PROGRAM EM8000
VAR	
	_control	: StewartControl;
	UdpIO		: UdpClient(3232258590, 50030, 50040, SIZEOF(_control), ADR(_control), SIZEOF(feedback), ADR(feedback));
	
	Pi 			: REAL := 3.141592653589793;
END_VAR

VAR_INPUT
	control		: StewartControl;
END_VAR

VAR_OUTPUT
	feedback	: StewartFeedback;
END_VAR



// Assign c0ntrol to local _control
_control.CMND := control.CMND;

// Addd maximum limit to udp input _control
_control.X_EXTRA 		:= LIMIT(-0.6, control.X_EXTRA, 0.6);
_control.Y_EXTRA 		:= LIMIT(-0.6, control.Y_EXTRA, 0.6);
_control.Z_EXTRA 		:= LIMIT(-0.6, control.Z_EXTRA, 0.6);

_control.PSI_EXTRA 		:= LIMIT(-10.0/180.0*Pi, control.PSI_EXTRA, 10.0/180.0*Pi);
_control.THETA_EXTRA 	:= LIMIT(-10.0/180.0*Pi, control.THETA_EXTRA, 10.0/180.0*Pi);
_control.PHI_EXTRA 		:= LIMIT(-10.0/180.0*Pi, control.PHI_EXTRA, 10.0/180.0*Pi);

_control.COUNT 			:= _control.COUNT + 1;

UdpIO();

END_PROGRAM

(* stored: Version 1.1.0.1, ProductVersion 3.1.4020.12
   POU EM8000: Id {c87bca3c-ddc6-4566-91d0-aa31a9002397}, SpecialFunc None *)
